FUNCTION_BLOCK AX_TO_AX2 (* Composite FB for convert unidirectional AX to bidirectional AX2 *)
  (* Standard: 61499-2; Function: AX_IN publishes its value onto the outgoing (EO1) side of AX2_BIDIR. Whatever AX2_BIDIR receives on its incoming (EI1) side is forwarded out again as a plain unidirectional signal via AX_OUT.; Description: Copyright (c) 2026 HR Agrartechnik GmbH This program and the accompanying materials are made available under the terms of the Eclipse Public License 2.0 which is available at https://www.eclipse.org/legal/epl-2.0/ SPDX-License-Identifier: EPL-2.0 *)
  (* Version 1.0, 2026-08-31, Franz Höpfinger, HR Agrartechnik GmbH, Initial Version *)
  PACKAGE adapter::conversion::bidirectional;
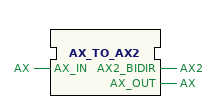
  SOCKETS
    AX_IN : adapter::types::unidirectional::AX; (* Adapter Input: unidirectional source *)
  END_SOCKETS
  PLUGS
    AX2_BIDIR : adapter::types::bidirectional::AX2; (* Adapter Output: bidirectional tap, outgoing side driven by AX_IN, incoming side forwarded to AX_OUT *)
    AX_OUT : adapter::types::unidirectional::AX; (* Adapter Output: mirrors AX2_BIDIR's incoming (request) side *)
  END_PLUGS
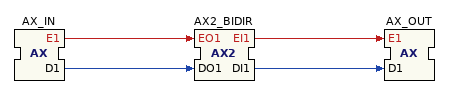
  EVENT_CONNECTIONS
    AX_IN.E1 TO AX2_BIDIR.EO1;
    AX2_BIDIR.EI1 TO AX_OUT.E1;
  END_CONNECTIONS
  DATA_CONNECTIONS
    AX_IN.D1 TO AX2_BIDIR.DO1;
    AX2_BIDIR.DI1 TO AX_OUT.D1;
  END_CONNECTIONS
END_FUNCTION_BLOCK
